(* IEC 61131-3 sources: Industry-PLC-LLM/data/PLCBEAD_repo/PLCBEAD_PLCEmbed-main/PLC-BEAD/Source/GEB/LEAP_DAY, 1 file *)

(* ---- LEAP_DAY.ST ---- *)
FUNCTION LEAP_DAY:BOOL

	VAR_INPUT
		IDATE :	UDINT;
	END_VAR

	LEAP_DAY  := IDATE MOD UDINT#126230400 = UDINT#68169600;

END_FUNCTION

PROGRAM program0
	VAR
		IDATE :	UDINT;
		OUT : BOOL;
	END_VAR

	OUT := LEAP_DAY(IDATE);
END_PROGRAM
